// TwinCAT 3 PLC project Untitled1
// ProgramVersion: 3.1.4023.0
// libraries:
//   Tc2_MC2, * (Beckhoff Automation GmbH)
//   Tc2_MC2_Drive, * (Beckhoff Automation GmbH)
//   Tc2_SerialCom, * (Beckhoff Automation GmbH)
//   Tc2_Standard, * (Beckhoff Automation GmbH)
//   Tc2_System, * (Beckhoff Automation GmbH)
//   Tc3_Module, * (Beckhoff Automation GmbH)
// project tree:
//   / ComTask.TcTTO (not stored), PlcTask.TcTTO
//   GVLs/GVLs/ GVL.TcGVL, GVL_IO.TcGVL, GVL_ResearchData.TcGVL, GVL_VAR.TcGVL, ReadMe.TcGVL (not stored)
//   POUs/ FB_Analog.TcPOU, F_ScalAnalogOut.TcPOU, MAIN.TcPOU, P_AP1_Calibrartion.TcPOU, P_ComEL6001.TcPOU (not stored), P_CP1_Enable.TcPOU, P_MI1_OnOff.TcPOU, P_AP1_OnOff.TcPOU, P_Outputs_Manual.TcPOU, P_Set_Research_Data.TcPOU, P_PP1_Ctrl_Manual.TcPOU, P_AP1_Ctrl_Manual.TcPOU, P_Read_Research_Data.TcPOU
//   POUs/POUs/ FB_Drive.TcPOU (not stored), FB_Mixer1_2.TcPOU (not stored)
// real-time tasks:
//   TASK PlcTask: cycle T#10ms, priority 20, ADS port 350
//   TASK ComTask: cycle T#10ms, priority 21, ADS port 351
// motion (NC):
//   TASK NC-Task 1 SAF: cycle T#2ms, priority 4, ADS port 501
//   TASK NC-Task 1 SVB: cycle T#10ms, priority 8, ADS port 511
//   AXIS Mixer 1 (id 2)
//     General: UnitName=°, UnitFlags=#x00000004
//     Dynamic: Acceleration=7443.34, Deceleration=7443.34, Jerk=22330
//     Velo: RefSearch=49.6222741699219, RefSync=49.6222741699219, SlowManual=248.111370849609, FastManual=1488.66822509766, Fast=4962.22741699219, Maximum=4962.23
//     OtherSettings: AllowMotionCmdToSlave=true
//     encoder EncType=8
//       EncPara: ScaleFactorNumerator=45, ScaleFactorDenominator=1048576, Offset=-131121.7408, Inverse=true, MaxCount=#x007fffff, ReferenceSystem=2
//     drive DrvType=9
//       DrvPara: Inverse=true, MaxCount=#xffffffff, DriveControlDWord=#x00030100
//         Analog: VeloReferenz=5458.45015869141, VeloScale=1.02400649589962, ScaleFactorActTorque=0.1
//         TimeComp: TaskDelayCycles=1
//     controller CtrType=1
//       CtrPara: PriorControlFactor=1
//         Observer: BandWidth=20
//   AXIS Mixer 2 (id 3)
//     General: UnitName=°, UnitFlags=#x00000004
//     Dynamic: Acceleration=7443.34112548828, Deceleration=7443.34112548828, Jerk=22330.0233764648
//     Velo: RefSearch=49.6222741699219, RefSync=49.6222741699219, SlowManual=248.111370849609, FastManual=1488.66822509766, Fast=4962.22741699219, Maximum=4962.22741699219
//     OtherSettings: AllowMotionCmdToSlave=true
//     encoder EncType=8
//       EncPara: ScaleFactorNumerator=45, ScaleFactorDenominator=1048576, MaxCount=#x007fffff, ReferenceSystem=2
//     drive DrvType=9
//       DrvPara: MaxCount=#xffffffff, DriveControlDWord=#x00030100
//         Analog: VeloReferenz=5458.45015869141, VeloScale=1.02400649589962, ScaleFactorActTorque=0.1
//         TimeComp: TaskDelayCycles=1
//     controller CtrType=1
//       CtrPara: PriorControlFactor=1
//         Observer: BandWidth=20
// I/O:
//   DEVICE Device 1 (EtherCAT), AmsNetId 172.17.147.1.3.1
//     Term 1 (EK1200) [EK1200-5000 EtherCAT Power supply (2A E-Bus)]
//       Term 2 (EL1008) 30K3 [EL1008 8Ch. Dig. Input 24V, 3ms]
//       Term 3 (EL1008) 30K3.1 [EL1008 8Ch. Dig. Input 24V, 3ms]
//       Term 10 (EL1008) new [EL1008 8Ch. Dig. Input 24V, 3ms]
//       Term 4 (EL2008) 30K4 [EL2008 8Ch. Dig. Output 24V, 0.5A]
//       Term 5 (EL2008) 30K5 [EL2008 8Ch. Dig. Output 24V, 0.5A]
//       Term 12 (EL2008) new [EL2008 8Ch. Dig. Output 24V, 0.5A]
//       Term 13 (EL3022) new [EL3022 2Ch. Ana. Input 4-20mA DIFF]
//       Term 14 (EL3202) new [EL3202 2Ch. Ana. Input PT100 (RTD)]
//       Term 6 (EL3255) 30K5.1 [EL3255 5Ch. potentiometer measurement with sensor supply]
//       Term 7 (EL4134) 30K6 [EL4134 4Ch. Ana. Output -10/+10V, 16bit]
//       Term 8 (EL6001) [EL6001 Interface (RS232)]
//       Term 15 (EL6631) new [EL6631 PROFINET IO Controller]
//       Term 9 (EL9011) [EL9011 End Terminal]
//   DEVICE Device 4 (EtherCAT), AmsNetId 172.17.147.1.5.1
//     Drive 11 (AX5206-0000-0213) [AX5206-0000-0213 EtherCAT Drive (SoE, 2 Ch.)]
// variable links:
//   NC-Task 1 SAF/Axes/Mixer 1 <-> Device 4 (EtherCAT)/Drive 11 (AX5206-0000-0213)
//     Drive/Inputs/In/nDataIn1 <-> AT 1/Following distance
//     Drive/Inputs/In/nDcOutputTime <-> InfoData/DcOutputShift
//     Drive/Inputs/In/nState1 <-> AT 1/Drive status word @bit 8
//     Drive/Inputs/In/nState2 <-> AT 1/Drive status word
//     Drive/Inputs/In/nState4 @bit 1 <-> WcState/InputToggle
//     Drive/Inputs/In/nState4 <-> WcState/WcState
//     Drive/Outputs/Out/nCtrl1 <-> MDT 1/Master control word @bit 8
//     Drive/Outputs/Out/nDataOut1 <-> MDT 1/Position command value
//     Enc/Inputs/In/nDataIn1 <-> AT 1/Position feedback 1 value
//     Enc/Inputs/In/nDcInputTime <-> InfoData/DcInputShift
//     Enc/Inputs/In/nState4 @bit 1 <-> WcState/InputToggle
//     Enc/Inputs/In/nState4 <-> WcState/WcState
//   NC-Task 1 SAF/Axes/Mixer 2 <-> Device 4 (EtherCAT)/Drive 11 (AX5206-0000-0213)
//     Drive/Inputs/In/nDataIn1 <-> AT 2/Following distance
//     Drive/Inputs/In/nDcOutputTime <-> InfoData/DcOutputShift
//     Drive/Inputs/In/nState1 <-> AT 2/Drive status word @bit 8
//     Drive/Inputs/In/nState2 <-> AT 2/Drive status word
//     Drive/Inputs/In/nState4 @bit 1 <-> WcState/InputToggle
//     Drive/Inputs/In/nState4 <-> WcState/WcState
//     Drive/Outputs/Out/nCtrl1 <-> MDT 2/Master control word @bit 8
//     Drive/Outputs/Out/nDataOut1 <-> MDT 2/Position command value
//     Enc/Inputs/In/nDataIn1 <-> AT 2/Position feedback 1 value
//     Enc/Inputs/In/nDcInputTime <-> InfoData/DcInputShift
//     Enc/Inputs/In/nState4 @bit 1 <-> WcState/InputToggle
//     Enc/Inputs/In/nState4 <-> WcState/WcState
//   Untitled1/Untitled1 Instance <-> Device 1 (EtherCAT)/Term 1 (EK1200)/Term 2 (EL1008) 30K3
//     ComTask Inputs/GVL_IO.ib_CC1_Button_Mode_Laptop <-> Channel 8/Input
//     ComTask Inputs/GVL_IO.ib_CP1_Ready <-> Channel 3/Input
//     PlcTask Inputs/GVL_IO.ib_AP1_No_Error <-> Channel 6/Input
//     PlcTask Inputs/GVL_IO.ib_AP1_Ready <-> Channel 5/Input
//     PlcTask Inputs/GVL_IO.ib_CC1_Button_Reset <-> Channel 7/Input
//     PlcTask Inputs/GVL_IO.ib_CC1_Safety_Ready <-> Channel 1/Input
//     PlcTask Inputs/GVL_IO.ib_CP1_Drive_Error <-> Channel 4/Input
//     PlcTask Inputs/GVL_IO.ib_CP1_Safety_Grid_Mounted <-> Channel 2/Input
//   Untitled1/Untitled1 Instance <-> Device 1 (EtherCAT)/Term 1 (EK1200)/Term 3 (EL1008) 30K3.1
//     ComTask Inputs/GVL_IO.ib_PP1_Button_Not_Off <-> Channel 5/Input
//     ComTask Inputs/GVL_IO.ib_PP1_Button_On <-> Channel 4/Input
//     PlcTask Inputs/GVL_IO.ib_AP1_Button_Not_Off <-> Channel 7/Input
//     PlcTask Inputs/GVL_IO.ib_AP1_Button_On <-> Channel 6/Input
//     PlcTask Inputs/GVL_IO.ib_CC1_Button_Mode_Manual <-> Channel 1/Input
//     PlcTask Inputs/GVL_IO.ib_MI1_Button_Not_Off <-> Channel 3/Input
//     PlcTask Inputs/GVL_IO.ib_MI1_Button_On <-> Channel 2/Input
//   Untitled1/Untitled1 Instance <-> Device 1 (EtherCAT)/Term 1 (EK1200)/Term 4 (EL2008) 30K4
//     PlcTask Outputs/GVL_IO.ob_AP1_Pressure_Ok <-> Channel 7/Output
//     PlcTask Outputs/GVL_IO.ob_AP1_Pulse <-> Channel 8/Output
//     PlcTask Outputs/GVL_IO.ob_AP1_Start <-> Channel 6/Output
//     PlcTask Outputs/GVL_IO.ob_CC1_Safety_Reset <-> Channel 1/Output
//     PlcTask Outputs/GVL_IO.ob_CP1_Backward <-> Channel 5/Output
//     PlcTask Outputs/GVL_IO.ob_CP1_Forward <-> Channel 4/Output
//     PlcTask Outputs/GVL_IO.ob_CP1_Start <-> Channel 3/Output
//     PlcTask Outputs/GVL_IO.ob_CP1_Stop <-> Channel 2/Output
//   Untitled1/Untitled1 Instance <-> Device 1 (EtherCAT)/Term 1 (EK1200)/Term 5 (EL2008) 30K5
//     PlcTask Outputs/GVL_IO.ob_AP1_Not_Empty <-> Channel 1/Output
//     PlcTask Outputs/GVL_IO.ob_AP1_Power_On <-> Channel 2/Output
//   Untitled1/Untitled1 Instance <-> Device 1 (EtherCAT)/Term 1 (EK1200)/Term 6 (EL3255) 30K5.1
//     ComTask Inputs/GVL_IO.in_AP1_Poti_Speed <-> AI Standard Channel 3/Value
//     ComTask Inputs/GVL_IO.in_PP1_Poti_Speed <-> AI Standard Channel 2/Value
//     PlcTask Inputs/GVL.nInputSpare1 <-> AI Standard Channel 4/Value
//     PlcTask Inputs/GVL.nInputSpare2 <-> AI Standard Channel 5/Value
//     PlcTask Inputs/GVL_IO.in_MI1_Poti_Speed <-> AI Standard Channel 1/Value
//   Untitled1/Untitled1 Instance <-> Device 1 (EtherCAT)/Term 1 (EK1200)/Term 7 (EL4134) 30K6
//     PlcTask Outputs/GVL_IO.on_AP1_Speed <-> AO Output Channel 2/Analog output
//     PlcTask Outputs/GVL_IO.on_CP1_Speed <-> AO Output Channel 1/Analog output
//   Untitled1/Untitled1 Instance <-> Device 1 (EtherCAT)/Term 1 (EK1200)/Term 8 (EL6001)
//     ComTask Inputs/GVL.stIn_EL6001/D <-> COM Inputs/Data In 0
//     ComTask Inputs/GVL.stIn_EL6001/D @bit {8..168 step 8} <-> COM Inputs/Data In {1..21}  (21 links)
//     ComTask Inputs/GVL.stIn_EL6001/Status <-> COM Inputs/Status
//     ComTask Outputs/GVL.stOut_EL6001/Ctrl <-> COM Outputs/Ctrl
//     ComTask Outputs/GVL.stOut_EL6001/D <-> COM Outputs/Data Out 0
//     ComTask Outputs/GVL.stOut_EL6001/D @bit {8..168 step 8} <-> COM Outputs/Data Out {1..21}  (21 links)
//   Untitled1/Untitled1 Instance <-> Device 4 (EtherCAT)/Drive 11 (AX5206-0000-0213)
//     PlcTask Inputs/GVL.in_MID1_ActAbsCurrent <-> AT 1/Actual absolute current
//     PlcTask Inputs/GVL.in_MID2_ActAbsCurrent <-> AT 2/Actual absolute current
//     PlcTask Inputs/GVL.in_MID1_ActMotorTemperature <-> AT 1/Motor temperature
//     PlcTask Inputs/GVL.in_MID2_ActMotorTemperature <-> AT 2/Motor temperature
//   Untitled1/Untitled1 Instance <-> NC-Task 1 SAF/Axes/Mixer 1
//     PlcTask Inputs/GVL.Axis_Mixer1.NcToPlc <-> Outputs/ToPlc
//     PlcTask Outputs/GVL.Axis_Mixer1.PlcToNc <-> Inputs/FromPlc
//   Untitled1/Untitled1 Instance <-> NC-Task 1 SAF/Axes/Mixer 2
//     PlcTask Inputs/GVL.Axis_Mixer2.NcToPlc <-> Outputs/ToPlc
//     PlcTask Outputs/GVL.Axis_Mixer2.PlcToNc <-> Inputs/FromPlc

CONFIGURATION Untitled1
    RESOURCE PLC ON TwinCAT3
        TASK PlcTask(INTERVAL := T#10ms, PRIORITY := 20);
        PROGRAM MAIN WITH PlcTask : MAIN;
    END_RESOURCE
END_CONFIGURATION

// ---- GVLs/GVLs/GVL.TcGVL
{attribute 'qualified_only'}
VAR_GLOBAL
	
	
	//
	// Data Communication RS-232
	TxBufferEL								: ComBuffer;
	RxBufferEL								: ComBuffer;
	
			
	//
	// Data Communication Axis Mixers

	//
	// Mixer drive A // 16.09.2021 PF
	Axis_Mixer1 							: AXIS_REF;
	f_MID1_ActCurrent: REAL;
	f_MID1_ActTorque: REAL;
	in_MID1_ActAbsCurrent AT %I*: INT;
	in_MID1_ActMotorTemperature AT %I* :INT; // 220817 weiting added
	
	//
	// Mixer drive B // 16.09.2021 PF
	Axis_Mixer2 							: AXIS_REF;
	f_MID2_ActCurrent: REAL;
	f_MID2_ActTorque: REAL;
	in_MID2_ActAbsCurrent AT %I*: INT;
	in_MID2_ActMotorTemperature AT %I* :INT; // 220817 weiting added
	
	//
	// Control Input Speed
	fControlMixerPumpSpeed					: REAL; 
	fControlPeristalticPumpSpeed			: REAL; 
	fControlDosingPumpSpeed					: REAL; 
	fInputSpare1							: REAL; 
	fInputSpare2							: REAL; 
	
	//
	// Output Speed
	fConcretePumpSpeed						: REAL;
	fDosingPumpSpeed						: REAL;
	fOutputSpare1							: REAL;
	fOutputSpare2							: REAL;
	
	
	//
	//Hardware Input
	bSafetyIO						AT %I*	: BOOL;
	// bConcretePumpSafetyGridMounted	AT %I*	: BOOL;
	// bConcretePumpReady				AT %I*	: BOOL;
	// bConcretePumpFcError				AT %I*	: BOOL;
	bDosingPumpReady				AT %I*	: BOOL;
	bDosingPumpNoError				AT %I*	: BOOL;
	bControlResetSafety				AT %I*	: BOOL;
	bControlLaptop					AT %I*	: BOOL;
	bControlManual					AT %I*	: BOOL;	
	nControlMixerPumpOn				AT %I*	: BOOL; 
	nControlMixerPumpOff			AT %I*	: BOOL; 
	nControlConcretPumpOn			AT %I*	: BOOL; 
	nControlConcretPumpOff			AT %I*	: BOOL; 
	nControlDosingPumpOn			AT %I*	: BOOL; 
	nControlDosingPumpOff			AT %I*	: BOOL; 
	bInputSpare1					AT %I*	: BOOL;
		
	nControlMixerPumpSpeed			AT %I*	: INT; 
	// nControlPeristalticPumpSpeed	AT %I*	: INT; 
	nControlDosingPumpSpeed			AT %I*	: INT; 
	nInputSpare1					AT %I*	: INT; 
	nInputSpare2					AT %I*	: INT; 

	
	//
	//Hardware Output
	bResetSafety					AT %Q*	: BOOL;
	// bConcretePumpOn					AT %Q*	: BOOL;
	// bConcretePumpOff					AT %Q*	: BOOL;
	// bConcretePumpForwardOn			AT %Q*	: BOOL;
	// bConcretePumpBackwardOn			AT %Q*	: BOOL;
	bDosingPumpDosingHighLow		AT %Q*	: BOOL;
	bDosingPumpNoFastStop			AT %Q*	: BOOL;
	bDosingPumpDosingAmount			AT %Q*	: BOOL;
	bOutputSpare1					AT %Q*	: BOOL;
	bOutputSpare2					AT %Q*	: BOOL;
	bOutputSpare3					AT %Q*	: BOOL;
	bOutputSpare4					AT %Q*	: BOOL;
	bOutputSpare5					AT %Q*	: BOOL;
	bOutputSpare6					AT %Q*	: BOOL;
	bOutputSpare7					AT %Q*	: BOOL;
	bOutputSpare8					AT %Q*	: BOOL;
	
	// nConcretePumpSpeed				AT %Q*	: INT;
	nDosingPumpSpeed				AT %Q*	: INT;
	nOutputSpare1					AT %Q*	: INT;
	nOutputSpare2					AT %Q*	: INT;
	
	
	//
	//Hardware RS-232
	stIn_EL6001 					AT %I*	: EL6inData22B;	
	stOut_EL6001 					AT %Q*	: EL6outData22B;
	
END_VAR

// ---- GVLs/GVLs/GVL_IO.TcGVL
{attribute 'qualified_only'}
VAR_GLOBAL
//***********************************************************************************
//
// ETH Zürich / Robotic Fabrication Lab
// HIB C 13 / Stefano-Franscini-Platz 1
// CH-8093 Zürich
// 
// ***********************************************************************************
// 
// PROJECT     :  A061 Inline Mixer
// 
// FUNCTION    :  Global Varable In and Outputs
// 
// AUTHOR      :  Fabio Scotto / Philippe Fleischmann
// 
// EMAIL       :  scotto@arch.ethz.ch / fleischmann@arch.ehtz.ch
// 
// Copyright   :  ETH Zürich (CH) 2020
//
// ***********************************************************************************

//
// Inputs

//
// Concrete Controller 1
ib_CC1_Safety_Ready AT %I*: BOOL;
ib_CC1_Button_Mode_Manual AT %I*: BOOL;
ib_CC1_Button_Mode_Laptop AT %I*: BOOL;
ib_CC1_Button_Reset AT %I*: BOOL;
//
// Concrete Pump 1
ib_CP1_Drive_Error AT %I*: BOOL;
ib_CP1_Ready AT %I*: BOOL;
ib_CP1_Safety_Grid_Mounted AT %I*: BOOL;
in_CP1_Tube_Pressure_Sensor AT %I*: INT;
in_CP1_Tube_Temperature_Sensor AT %I*: INT;

//
// Peristaltic Pump 1
ib_PP1_Button_On AT %I*: BOOL;
ib_PP1_Button_Not_Off AT %I*: BOOL;
in_PP1_Poti_Speed AT %I*	: INT; 

//
// Accelerator Pump 1
ib_AP1_Button_On AT %I*: BOOL;
ib_AP1_Button_Not_Off AT %I*: BOOL;
ib_AP1_Ready AT %I*: BOOL;
ib_AP1_No_Error AT %I*: BOOL;
in_AP1_Poti_Speed AT %I*	: INT; 

//
// Mixer 1
ib_MI1_Button_On AT %I*: BOOL;
ib_MI1_Button_Not_Off AT %I*: BOOL;
in_MI1_Poti_Speed AT %I*	: INT; 

//
// Outputs

//
// Concrete Controller 1
ob_CC1_Safety_Reset AT %Q*: BOOL;

//
// Concrete Pump 1
ob_CP1_Start AT %Q*: BOOL;
ob_CP1_Stop AT %Q*: BOOL;
ob_CP1_Forward AT %Q*: BOOL;
ob_CP1_Backward AT %Q*: BOOL;

on_CP1_Speed AT %Q*: INT;

//
// Accelerator Pump 1
ob_AP1_Power_On AT %Q*: BOOL;
ob_AP1_Start AT %Q*: BOOL;
ob_AP1_Pressure_Ok AT %Q*: BOOL;
ob_AP1_Not_Empty AT %Q*: BOOL;
ob_AP1_Pulse AT %Q*: BOOL;

on_AP1_Speed AT %Q*: INT;


END_VAR

// ---- GVLs/GVLs/GVL_ResearchData.TcGVL
{attribute 'qualified_only'}
VAR_GLOBAL
//***********************************************************************************
//
// ETH Zürich / Robotic Fabrication Lab
// HIB C 13 / Stefano-Franscini-Platz 1
// CH-8093 Zürich
// 
// ***********************************************************************************
// 
// PROJECT     :  A061 Inline Mixer
// 
// FUNCTION    :  Global Varable to collect all research data
// 
// AUTHOR      :  Seyma Gürel / Philippe Fleischmann
// 
// EMAIL       :  scotto@arch.ethz.ch / fleischmann@arch.ehtz.ch
// 
// Copyright   :  ETH Zürich (CH) 2021
//
// ***********************************************************************************


// ***********************************************************************************
// Process inputs
// ***********************************************************************************

//
// Maximal speed for mixer [°/s]  
f_RED_Control_Speed : LREAL;					// [°/s]

//
// Accelerator Pump
b_RED_Acceleration_Pump_Calibration_On: BOOL;
n_RED_Acceleration_Pump_Calibration_Speed: INT;
n_RED_Acceleration_Pump_Calibration_Time: TIME;
f_RED_Acceleration_Pump_Mass: REAL;             // [g/min]
f_RED_Acceleration_Pump_Density: REAL;          // [g/ml]
n_RED_Acceleration_Pump_Flowrate: REAL;         // [ml/min]

//
// Concrete Pump
b_RED_Concrete_Pump_Forward_On: BOOL;
b_RED_Concrete_Pump_Backward_On: BOOL;
n_RED_Concrete_Pump_Speed: INT;					// [ 0..75rpm ]
		

// ***********************************************************************************
// Process outpus
// ***********************************************************************************

//
// Status mixer
b_RED_Status_On : BOOL;
f_RED_Status_Speed_Overide : LREAL;
f_RED_Status_Speed_Motor_1 : LREAL;
f_RED_Status_Speed_Motor_2 : LREAL;
f_RED_Status_Torque_Motor_1 : REAL;				// [Nm]
f_RED_Status_Torque_Motor_2 : REAL;				// [Nm]

// Weiting added 220817 
f_RED_Status_Temperature_Motor_1 : REAL; // [°C] 
f_RED_Status_Temperature_Motor_2 : REAL; // [°C] 

//
// Accelerator Pump
n_RED_Status_Acceleration_Pump_Flowrate: INT;          // [ml/min]
f_RED_Status_Acceleration_Pump_Max_Flowrate_ml_per_min: REAL;           // [ml/min]

END_VAR

// ---- GVLs/GVLs/GVL_VAR.TcGVL
{attribute 'qualified_only'}
VAR_GLOBAL
//***********************************************************************************
//
// ETH Zürich / Robotic Fabrication Lab
// HIB C 13 / Stefano-Franscini-Platz 1
// CH-8093 Zürich
// 
// ***********************************************************************************
// 
// PROJECT     :  A061 Inline Mixer
// 
// FUNCTION    :  Global Varable In and Outputs
// 
// AUTHOR      :  Fabio Scotto / Philippe Fleischmann
// 
// EMAIL       :  scotto@arch.ethz.ch / fleischmann@arch.ehtz.ch
// 
// Copyright   :  ETH Zürich (CH) 2020
//
// ***********************************************************************************

//
// Concrete Controller 1

//
// Concrete Pump 1

//
// Peristaltic Pump 1

//
// Accelerator Pump 1
b_AP1_Run : BOOL;
f_AP1_Override : LREAL; 

//
// Mixer 1
b_MI1_ReadToDrive : BOOL;
b_MI1_Run : BOOL;
f_MI1_Override : LREAL; 
f_MI1_MaxSpeed : LREAL;
f_MI1_ActSpeedM1 : LREAL;
f_MI1_ActSpeedM2 : LREAL;

END_VAR

// ---- POUs/MAIN.TcPOU
PROGRAM MAIN
VAR	

	fb_MC_SetPosition		:FB_SoEAX5000SetPositionOffset;
	pos:real;
	Mixer1_2		: FB_Mixer1_2;
	Analog			: FB_Analog;

	SafetyReset 	: bool;
	b_Enable		: BOOL;
	b_Reset			: BOOL;


	
	Test : MC_ReadStatus;
END_VAR

//***********************************************************************************
//
// ETH Zürich / Robotic Fabrication Lab
// HIB C 13 / Stefano-Franscini-Platz 1
// CH-8093 Zürich
// 
// ***********************************************************************************
// 
// PROJECT     :  A061 Inline Mixer
// 
// FUNCTION    :  MAIN Programm
// 
// AUTHOR      :  Mathias Suter
// 
// EMAIL       :  mathias.suter@solinaut.ch
// 
// Copyright   :  ETH Zürich (CH) 2021
//
// ***********************************************************************************


//
// Mode selector 
//P_ModeSelector();

//
// Set research data 
P_Set_Research_Data();

//
// Acceleration Pump 1 On/off 
P_AP1_Calibrartion();

//
// Check for Acceleration Pump 1 state
IF GVL_ResearchData.b_RED_Acceleration_Pump_Calibration_On=FALSE THEN
	//
	// Acceleration Pump 1 On/off 
	P_AP1_OnOff();
END_IF

//
// Temporary scaling of the poti for the mixer override  
GVL_VAR.f_MI1_Override:=100.0 / 32767 * GVL_IO.in_MI1_Poti_Speed;

//
// Peristaltic Pump 1 manual control 
//P_PP1_Ctrl_Manual();

//
// Mixer On/Off 
P_MI1_OnOff();

//
// Temporary scaling of the poti for the mixer override  
GVL_VAR.f_MI1_Override:=100.0 / 32767 * GVL_IO.in_MI1_Poti_Speed;

//
// Mixer 1 + 2
Mixer1_2(
	Mixer1			:= GVL.Axis_Mixer1,
 	Mixer2			:= GVL.Axis_Mixer2,
	f_Velocity		:= GVL_VAR.f_MI1_MaxSpeed,
	b_JogForward	:= FALSE,
	b_JogBackwards	:= GVL_VAR.b_MI1_Run,
 	b_Enable		:= GVL_IO.ib_CC1_Button_Mode_Manual AND GVL_IO.ib_CC1_Safety_Ready,	
 	b_Reset			:= GVL_IO.ib_CC1_Button_Reset,
	f_Override		:= GVL_VAR.f_MI1_Override);	
	(*
	fb_MC_SetPosition(
	Axis			:= GVL.Axis_Mixer2,
	memory			:= 1,
	Feedback		:= 0);*)
	
pos:=GVL.Axis_Mixer2.NcToPlc.ModuloActPos;


//
GVL.f_MID1_ActCurrent:=GVL.in_MID1_ActAbsCurrent * 5.9 / 1000;
GVL.f_MID1_ActTorque:=GVL.f_MID1_ActCurrent * 1.4 * 8; // Torque constante / Gear transaltion

GVL.f_MID2_ActCurrent:=gvl.in_MID2_ActAbsCurrent * 5.9 / 1000;
GVL.f_MID2_ActTorque:=GVL.f_MID2_ActCurrent * 1.4 * 8; // Torque constante / Gear transaltion

//
// Write global variable for mixer ready to drive
GVL_VAR.b_MI1_ReadToDrive:=Mixer1_2.b_ReadyToDrive;
	
// 
// Reset 
GVL_IO.ob_CC1_Safety_Reset:=GVL_IO.ib_CC1_Button_Reset;
 	
// GVL.bResetSafety	:= safetyReset;


//
// Concrete pump
P_CP1_Enable();
	
// Analog();

//
// Outputs
P_Outputs_Manual();

//
// Read researchs data 
P_Read_Research_Data();

END_PROGRAM

// ---- POUs/FB_Analog.TcPOU
FUNCTION_BLOCK FB_Analog
VAR_INPUT
END_VAR
VAR_OUTPUT
END_VAR
VAR
END_VAR

//***********************************************************************************
//
// ETH Zürich / Robotic Fabrication Lab
// HIB C 13 / Stefano-Franscini-Platz 1
// CH-8093 Zürich
// 
// ***********************************************************************************
// 
// PROJECT     :  ?? 
// 
// FUNCTION    :  Analog Calculation
// 
// AUTHOR      :  Mathias Suter
// 
// EMAIL       :  mathias.suter@solinaut.ch
// 
// Copyright   :  ETH Zürich (CH) 2021
//
// ***********************************************************************************


//
// Analog Inputs - Scale 0-100%
GVL.fControlMixerPumpSpeed := INT_TO_REAL(GVL.nControlMixerPumpSpeed) / 32767 * 100;			
//GVL.fControlPeristalticPumpSpeed := INT_TO_REAL(GVL.nControlPeristalticPumpSpeed) / 32767 * 100;			
GVL.fControlDosingPumpSpeed := INT_TO_REAL(GVL.nControlDosingPumpSpeed) / 32767 * 100;				
GVL.fInputSpare1 := INT_TO_REAL(GVL.nInputSpare1) / 32767 * 100;						
GVL.fInputSpare2 := INT_TO_REAL(GVL.nInputSpare2) / 32767 * 100;						
	

//
// Analog Outputs - Scale 0-100%
// GVL.nConcretePumpSpeed := REAL_TO_INT(GVL.fConcretePumpSpeed / 100 * 32767);				
GVL.nDosingPumpSpeed := REAL_TO_INT(GVL.fDosingPumpSpeed / 100 * 32767);					
GVL.nOutputSpare1 := REAL_TO_INT(GVL.fOutputSpare1 / 100 * 32767);						
GVL.nOutputSpare2 := REAL_TO_INT(GVL.fOutputSpare2 / 100 * 32767);

END_FUNCTION_BLOCK

// ---- POUs/P_Set_Research_Data.TcPOU
PROGRAM P_Set_Research_Data
VAR


END_VAR

//***********************************************************************************
//
// ETH Zürich / Robotic Fabrication Lab
// HIB C 13 / Stefano-Franscini-Platz 1
// CH-8093 Zürich
// 
// ***********************************************************************************
// 
// PROJECT     :  A061 Inline Mixer
// 
// FUNCTION    :  Set all research data for the process
// 
// AUTHOR      :  Seyma Gürel / Philippe Fleischmann
// 
// EMAIL       :  scotto@arch.ethz.ch / fleischmann@arch.ehtz.ch
// 
// Copyright   :  ETH Zürich (CH) 2021
//
// ***********************************************************************************


//
// Updating Mixer 1 max speed [°/s]
GVL_ResearchData.f_RED_Control_Speed:=720;
GVL_VAR.f_MI1_MaxSpeed:=GVL_ResearchData.f_RED_Control_Speed;

//
// Updating Acceleration Pump calibration values 
GVL_ResearchData.n_RED_Acceleration_Pump_Calibration_Speed:=32767;     // [raw date]
GVL_ResearchData.n_RED_Acceleration_Pump_Calibration_Time:=T#60000MS;   // [ms]
//GVL_ResearchData.f_RED_Acceleration_Pump_Mass:=342.0;                    // [g/min]
GVL_ResearchData.f_RED_Acceleration_Pump_Density:=2.047;               // [g/ml]

END_PROGRAM

// ---- POUs/P_AP1_Calibrartion.TcPOU
PROGRAM P_AP1_Calibrartion
VAR_INPUT
	//
	// INT 
	n_Step: INT := 0;	
END_VAR
VAR
	//
	// BOOL 
	b_Condition: BOOL;

	//
	// Timer
	t_AP1_Calibration_Time: TON; 
	
END_VAR

//***********************************************************************************
//
// ETH Zürich / Robotic Fabrication Lab
// HIB C 13 / Stefano-Franscini-Platz 1
// CH-8093 Zürich
// 
// ***********************************************************************************
// 
// PROJECT     :  A061 Inline Mixer
// 
// FUNCTION    :  Step chain for accelerator pump calibration
// 
// AUTHOR      :  Seyma Gürel / Philippe Fleischmann
// 
// EMAIL       :  sguerel@ethz.ch / fleischmann@arch.ehtz.ch
// 
// Copyright   :  ETH Zürich (CH) 2021
//
// ***********************************************************************************

//
// Initalization
IF n_Step=0 THEN
	//
	// Check condition 
	b_Condition:=TRUE;
	//
	// Do step
	IF b_Condition THEN
		b_Condition:=FALSE;
		n_Step:=10;
	END_IF
END_IF

//
// Wait for activating calibration
IF n_Step=10 THEN
	//
	// Check condition 
	b_Condition:= GVL_ResearchData.b_RED_Acceleration_Pump_Calibration_On;
	//
	// Do step
	IF b_Condition THEN
		b_Condition:=FALSE;
		n_Step:=20;
	END_IF
END_IF

//
// Wait for start 
IF n_Step=20 THEN
	//
	// Check condition 
	b_Condition:=GVL_IO.ib_AP1_Button_On;
	//
	// Do step
	IF b_Condition THEN
		b_Condition:=FALSE;
		n_Step:=30;
	END_IF
END_IF

//
// Run calibration until time is over 
IF n_Step=30 THEN
	//
	// Check condition 
	b_Condition:=t_AP1_Calibration_Time.Q; 
	//
	// Do step
	IF b_Condition THEN
		b_Condition:=FALSE;
		n_Step:=40;
	END_IF
END_IF

//
// Return to step 10 
IF n_Step=40 THEN
	//
	// Check condition 
	b_Condition:=TRUE;
	//
	// Do step
	IF b_Condition THEN
		b_Condition:=FALSE;
		//
		// Reset calibrarion on
		GVL_ResearchData.b_RED_Acceleration_Pump_Calibration_On:=FALSE;
		n_Step:=10;
	END_IF
END_IF

// ****************************************
// Timer
// ****************************************
t_AP1_Calibration_Time(
	IN:=n_Step=30,
	PT:=GVL_ResearchData.n_RED_Acceleration_Pump_Calibration_Time);

// ****************************************
// Reset
// ****************************************

IF GVL_ResearchData.b_RED_Acceleration_Pump_Calibration_On=FALSE THEN
  //
  // Rest step chain
  n_Step:=0;
END_IF

END_PROGRAM

// ---- POUs/P_AP1_OnOff.TcPOU
PROGRAM P_AP1_OnOff
VAR_INPUT
	//
	// INT 
	n_Step: INT := 0;	
END_VAR
VAR
	//
	// BOOL 
	b_Condition: BOOL;
	b_No_Emergency_Stop:BOOL :=TRUE;
	
END_VAR

//***********************************************************************************
//
// ETH Zürich / Robotic Fabrication Lab
// HIB C 13 / Stefano-Franscini-Platz 1
// CH-8093 Zürich
// 
// ***********************************************************************************
// 
// PROJECT     :  A061 Inline Mixer
// 
// FUNCTION    :  Step chain for accelerator pump on or off 
// 
// AUTHOR      :  Fabio Scotto / Philippe Fleischmann
// 
// EMAIL       :  scotto@arch.ethz.ch / fleischmann@arch.ehtz.ch
// 
// Copyright   :  ETH Zürich (CH) 2020
//
// ***********************************************************************************

//
// Ignore emergency stop
b_No_Emergency_Stop:=TRUE;

//
// Initalization
IF n_Step=0 THEN
	//
	// Check condition 
	b_Condition:=TRUE;
	//
	// Do step
	IF b_Condition THEN
		b_Condition:=FALSE;
		n_Step:=10;
	END_IF
END_IF

//
// Wait for start mixer
IF n_Step=10 THEN
	//
	// Check condition 
	b_Condition:= GVL_IO.ib_AP1_Ready AND GVL_IO.ib_AP1_Button_On;
	//
	// Do step
	IF b_Condition AND b_No_Emergency_Stop THEN
		b_Condition:=FALSE;
		n_Step:=20;
	END_IF
END_IF

//
// Reserve
IF n_Step=20 THEN
	//
	// Check condition 
	b_Condition:=TRUE;
	//
	// Do step
	IF b_Condition AND b_No_Emergency_Stop THEN
		b_Condition:=FALSE;
		n_Step:=30;
	END_IF
END_IF

//
// Run for mixer 
IF n_Step=30 THEN
	//
	// Check condition 
	b_Condition:= NOT GVL_IO.ib_AP1_Button_Not_Off OR NOT GVL_IO.ib_AP1_No_Error ;
	//
	// Do step
	IF b_Condition THEN
		b_Condition:=FALSE;
		n_Step:=40;
	END_IF
END_IF

//
// Reserve
IF n_Step=40 THEN
	//
	// Check condition 
	b_Condition:=TRUE;
	//
	// Do step
	IF b_Condition AND b_No_Emergency_Stop THEN
		b_Condition:=FALSE;
		n_Step:=50;
	END_IF
END_IF

//
// Return to step 10 
IF n_Step=50 THEN
	//
	// Check condition 
	b_Condition:=TRUE;
	//
	// Do step
	IF b_Condition THEN
		b_Condition:=FALSE;
		n_Step:=10;
	END_IF
END_IF

// ****************************************
// Write global variabls
// ****************************************

//
// Mixer run
GVL_VAR.b_AP1_Run:=n_Step=30;


// ****************************************
// Timer
// ****************************************

END_PROGRAM

// ---- POUs/P_MI1_OnOff.TcPOU
PROGRAM P_MI1_OnOff
VAR_INPUT
	//
	// INT 
	n_Step: INT := 0;	
END_VAR
VAR
	//
	// BOOL 
	b_Condition: BOOL;
	b_No_Emergency_Stop:BOOL :=TRUE;
	
END_VAR

//***********************************************************************************
//
// ETH Zürich / Robotic Fabrication Lab
// HIB C 13 / Stefano-Franscini-Platz 1
// CH-8093 Zürich
// 
// ***********************************************************************************
// 
// PROJECT     :  A061 Inline Mixer
// 
// FUNCTION    :  Step chain for mixer on or off 
// 
// AUTHOR      :  Fabio Scotto / Philippe Fleischmann
// 
// EMAIL       :  scotto@arch.ethz.ch / fleischmann@arch.ehtz.ch
// 
// Copyright   :  ETH Zürich (CH) 2020
//
// ***********************************************************************************

// Ignore emergency stop
b_No_Emergency_Stop:=TRUE;

//
// Initalization
IF n_Step=0 THEN
	//
	// Check condition 
	b_Condition:=TRUE;
	//
	// Do step
	IF b_Condition THEN
		b_Condition:=FALSE;
		n_Step:=10;
	END_IF
END_IF

//
// Wait for start mixer
IF n_Step=10 THEN
	//
	// Check condition 
	b_Condition:= GVL_VAR.b_MI1_ReadToDrive AND GVL_IO.ib_MI1_Button_On;
	//
	// Do step
	IF b_Condition AND b_No_Emergency_Stop THEN
		b_Condition:=FALSE;
		n_Step:=20;
	END_IF
END_IF

//
// Reserve
IF n_Step=20 THEN
	//
	// Check condition 
	b_Condition:=TRUE;
	//
	// Do step
	IF b_Condition AND b_No_Emergency_Stop THEN
		b_Condition:=FALSE;
		n_Step:=30;
	END_IF
END_IF

//
// Run for mixer 
IF n_Step=30 THEN
	//
	// Check condition 
	b_Condition:= NOT GVL_IO.ib_MI1_Button_Not_Off OR NOT GVL_VAR.b_MI1_ReadToDrive;
	//
	// Do step
	IF b_Condition THEN
		b_Condition:=FALSE;
		n_Step:=40;
	END_IF
END_IF

//
// Reserve
IF n_Step=40 THEN
	//
	// Check condition 
	b_Condition:=TRUE;
	//
	// Do step
	IF b_Condition AND b_No_Emergency_Stop THEN
		b_Condition:=FALSE;
		n_Step:=50;
	END_IF
END_IF

//
// Return to step 10 
IF n_Step=50 THEN
	//
	// Check condition 
	b_Condition:=TRUE;
	//
	// Do step
	IF b_Condition THEN
		b_Condition:=FALSE;
		n_Step:=10;
	END_IF
END_IF

// ****************************************
// Write global variabls
// ****************************************

//
// Mixer run
GVL_VAR.b_MI1_Run:=n_Step=30;


// ****************************************
// Timer
// ****************************************

END_PROGRAM

// ---- POUs/P_CP1_Enable.TcPOU
PROGRAM P_CP1_Enable
VAR_INPUT
	//
	// INT 
	n_Step: INT := 0;	
END_VAR
VAR
	//
	// BOOL 
	b_Condition: BOOL;
	b_No_Emergency_Stop:BOOL :=TRUE;

	//
	// Timer 
	t_CP1_Puls_Enable: TON;	
	t_CP1_Puls_Disable: TON;	
	
END_VAR

//***********************************************************************************
//
// ETH Zürich / Robotic Fabrication Lab
// HIB C 13 / Stefano-Franscini-Platz 1
// CH-8093 Zürich
// 
// ***********************************************************************************
// 
// PROJECT     :  A059 Aero Crete 
// 
// FUNCTION    :  Step chain for concrete pump enable 
// 
// AUTHOR      :  Nicolas Feihl / Philippe Fleischmann
// 
// EMAIL       :  feihl@arch.ethz.ch / fleischmann@arch.ehtz.ch
// 
// Copyright   :  ETH Zürich (CH) 2020
//
// ***********************************************************************************

// Ignore emergency stop
b_No_Emergency_Stop:=TRUE;

//
// Initalization
IF n_Step=0 THEN
	//
	// Check condition 
	b_Condition:=TRUE;
	//
	// Do step
	IF b_Condition THEN
		b_Condition:=FALSE;
		n_Step:=10;
	END_IF
END_IF

//
// Check grid mounted and no errors 
IF n_Step=10 THEN
	//
	// Check condition 
	b_Condition:= GVL_IO.ib_CP1_Safety_Grid_Mounted AND NOT GVL_IO.ib_CP1_Drive_Error;
	//
	// Do step
	IF b_Condition AND b_No_Emergency_Stop THEN
		b_Condition:=FALSE;
		n_Step:=20;
	END_IF
END_IF

//
// Send enable to pump
IF n_Step=20 THEN
	//
	// Check condition 
	b_Condition:=t_CP1_Puls_Enable.Q;
	//
	// Do step
	IF b_Condition AND b_No_Emergency_Stop THEN
		b_Condition:=FALSE;
		n_Step:=30;
	END_IF
END_IF

//
// Pump enabled checking for errors or grid removed
IF n_Step=30 THEN
	//
	// Check condition 
	b_Condition:= NOT GVL_IO.ib_CP1_Safety_Grid_Mounted OR GVL_IO.ib_CP1_Drive_Error;
	//
	// Do step
	IF b_Condition THEN
		b_Condition:=FALSE;
		n_Step:=40;
	END_IF
END_IF

//
// Send disable to pump
IF n_Step=40 THEN
	//
	// Check condition 
	b_Condition:=t_CP1_Puls_Disable.Q;
	//
	// Do step
	IF b_Condition AND b_No_Emergency_Stop THEN
		b_Condition:=FALSE;
		n_Step:=50;
	END_IF
END_IF

//
// Return to step 10 
IF n_Step=50 THEN
	//
	// Check condition 
	b_Condition:=TRUE;
	//
	// Do step
	IF b_Condition THEN
		b_Condition:=FALSE;
		n_Step:=10;
	END_IF
END_IF

// ****************************************
// Timer
// ****************************************
t_CP1_Puls_Enable(
	IN:=n_Step=20,
	PT:=T#200MS);

t_CP1_Puls_Disable(
	IN:=n_Step=40,
	PT:=T#200MS);

END_PROGRAM

// ---- POUs/P_Outputs_Manual.TcPOU
PROGRAM P_Outputs_Manual
VAR


END_VAR

//***********************************************************************************
//
// ETH Zürich / Robotic Fabrication Lab
// HIB C 13 / Stefano-Franscini-Platz 1
// CH-8093 Zürich
// 
// ***********************************************************************************
// 
// PROJECT     :  A061 Inline Mixer
// 
// FUNCTION    :  Outputs Manual Mode
// 
// AUTHOR      :  Fabio Scotto / Philippe Fleischmann
// 
// EMAIL       :  scotto@arch.ethz.ch / fleischmann@arch.ehtz.ch
// 
// Copyright   :  ETH Zürich (CH) 2020
//
// ***********************************************************************************


//
// Accelerator pump 1

//
// Power on
GVL_IO.ob_AP1_Power_On:=GVL_IO.ib_CC1_Button_Mode_Manual;

//
// Pressure okey always set to true
GVL_IO.ob_AP1_Pressure_Ok:=TRUE;

//
// Bucket not empty always set to true
GVL_IO.ob_AP1_Not_Empty:=TRUE;

//
// Pulse a preset amount not in use
GVL_IO.ob_AP1_Pulse:=FALSE;

//
// Start pump
IF 	   P_AP1_OnOff.n_Step=30 
	OR P_AP1_Calibrartion.n_Step=30
THEN
	//
	// Pump on
	GVL_IO.ob_AP1_Start:=TRUE;
ELSE
	//
	// Pump off
	GVL_IO.ob_AP1_Start:=FALSE;
END_IF

//
// Speed for pump
IF 	   P_AP1_Calibrartion.n_Step=20 
	OR P_AP1_Calibrartion.n_Step=30 
THEN
	//
	// Calibration Speed for pump
	GVL_IO.on_AP1_Speed:=GVL_ResearchData.n_RED_Acceleration_Pump_Calibration_Speed;
ELSE
	//
	// Process speed for pump
	GVL_IO.on_AP1_Speed:=F_ScalAnalogOut(
		n_Input:= REAL_TO_INT(GVL_ResearchData.n_RED_Acceleration_Pump_Flowrate),
		n_InMin:= 0, 
		n_InMax:= REAL_TO_INT(GVL_ResearchData.f_RED_Status_Acceleration_Pump_Max_Flowrate_ml_per_min), 
		n_OutMin:= 0, 
		n_OutMax:= 32767);
END_IF

// ***********************************************************************************
// Concrete Pump 1 
// ***********************************************************************************

//
// Start
IF  P_CP1_Enable.n_Step=20 THEN
	GVL_IO.ob_CP1_Start:=TRUE;
ELSE
	GVL_IO.ob_CP1_Start:=FALSE;
END_IF

//
// Stop
IF  P_CP1_Enable.n_Step=40 THEN
	GVL_IO.ob_CP1_Stop:=TRUE;
ELSE
	GVL_IO.ob_CP1_Stop:=FALSE;
END_IF

//
// Forward
GVL_IO.ob_CP1_Forward:=GVL_ResearchData.b_RED_Concrete_Pump_Forward_On;

//
// Backward
GVL_IO.ob_CP1_Backward:=GVL_ResearchData.b_RED_Concrete_Pump_Backward_On;

//
// Concrete pump speed  0 (0V) to 75 rpm (10V)
GVL_IO.on_CP1_Speed:=F_ScalAnalogOut(
	n_Input:=GVL_ResearchData.n_RED_Concrete_Pump_Speed, 
	n_InMin:=0, 
	n_InMax:=75, 
	n_OutMin:=0, 
	n_OutMax:=32767);

END_PROGRAM

// ---- POUs/F_ScalAnalogOut.TcPOU
FUNCTION F_ScalAnalogOut : INT
VAR_INPUT
	n_Input:INT;
	n_InMin:INT;
	n_InMax:INT;
	n_OutMin:INT;
	n_OutMax:INT;

END_VAR
VAR
	f_Input:REAL;
	f_InMin:REAL;
	f_InMax:REAL;
	f_OutMin:REAL;
	f_OutMax:REAL;
	f_DeltaIn:REAL;
	f_DeltaOut:REAL;
END_VAR

//
// Convert integer to real 
f_Input:=INT_TO_REAL(n_Input);
f_InMin:=INT_TO_REAL(n_InMin);
f_InMax:=INT_TO_REAL(n_InMax);
f_OutMin:=INT_TO_REAL(n_OutMin);
f_OutMax:=INT_TO_REAL(n_OutMax);
//
// Check plausibility 
IF f_InMax = f_InMin THEN	
	//
	// Not plausible output fix value
	F_ScalAnalogOut := 0;
ELSE	
	//
	// Plausible calculate output 
	f_DeltaIn:=f_InMax-f_InMin;
	f_DeltaOut:=f_OutMax-f_OutMin;
	F_ScalAnalogOut :=REAL_TO_INT((f_DeltaOut/f_DeltaIn)*(f_Input-f_InMin));	
END_IF

END_FUNCTION

// ---- POUs/P_Read_Research_Data.TcPOU
PROGRAM P_Read_Research_Data
VAR


END_VAR

//***********************************************************************************
//
// ETH Zürich / Robotic Fabrication Lab
// HIB C 13 / Stefano-Franscini-Platz 1
// CH-8093 Zürich
// 
// ***********************************************************************************
// 
// PROJECT     :  A061 Inline Mixer
// 
// FUNCTION    :  Read all research data for the process
// 
// AUTHOR      :  Seyma Gürel / Philippe Fleischmann
// 
// EMAIL       :  scotto@arch.ethz.ch / fleischmann@arch.ehtz.ch
// 
// Copyright   :  ETH Zürich (CH) 2021
//
// ***********************************************************************************


//
// Mixer run []
GVL_ResearchData.b_RED_Status_On:=GVL_VAR.b_MI1_Run;

//
// Mixer 1 speed override [%]
GVL_ResearchData.f_RED_Status_Speed_Overide:=GVL_VAR.f_MI1_Override;

//
// Mixer 1 current speed []
GVL_ResearchData.f_RED_Status_Speed_Motor_1:=GVL.Axis_Mixer1.NcToPlc.ActVelo;

//
// Mixer 1 current torque []
GVL_ResearchData.f_RED_Status_Torque_Motor_1:=GVL.f_MID1_ActTorque;

//
// Mixer 1 current motor temperature []
GVL_ResearchData.f_RED_Status_Temperature_Motor_1:=GVL.in_MID1_ActMotorTemperature *0.1; // weiting added 220817

//
// Mixer 2 current speed []
GVL_ResearchData.f_RED_Status_Speed_Motor_2:=GVL.Axis_Mixer1.NcToPlc.ActVelo;

//
// Mixer 2 current torque []
GVL_ResearchData.f_RED_Status_Torque_Motor_2:=GVL.f_MID2_ActTorque;

//
// Mixer 1 current motor temperature []
GVL_ResearchData.f_RED_Status_Temperature_Motor_2:=GVL.in_MID2_ActMotorTemperature *0.1; // weiting added 220817


//
// Accelration pump flowrate [ml/min]
GVL_ResearchData.f_RED_Status_Acceleration_Pump_Max_Flowrate_ml_per_min:=(GVL_ResearchData.f_RED_Acceleration_Pump_Mass/GVL_ResearchData.f_RED_Acceleration_Pump_Density);

END_PROGRAM

// ---- POUs/P_PP1_Ctrl_Manual.TcPOU
PROGRAM P_PP1_Ctrl_Manual
VAR
END_VAR

//***********************************************************************************
//
// ETH Zürich / Robotic Fabrication Lab
// HIB C 13 / Stefano-Franscini-Platz 1
// CH-8093 Zürich
// 
// ***********************************************************************************
// 
// PROJECT     :  A061 Inline Mixer
// 
// FUNCTION    :  Manual control of acceleration pump 1 
// 
// AUTHOR      :  Fabio Scotto / Philippe Fleischmann
// 
// EMAIL       :  scotto@arch.ethz.ch / fleischmann@arch.ehtz.ch
// 
// Copyright   :  ETH Zürich (CH) 2020
//
// ***********************************************************************************

//
// Place holder for manual control of the peristaltic pump 

;

END_PROGRAM

// ---- POUs/P_AP1_Ctrl_Manual.TcPOU
PROGRAM P_AP1_Ctrl_Manual

VAR

b_AP1_Error : BOOL;
b_AP1_Ready : BOOL;


END_VAR

//***********************************************************************************
//
// ETH Zürich / Robotic Fabrication Lab
// HIB C 13 / Stefano-Franscini-Platz 1
// CH-8093 Zürich
// 
// ***********************************************************************************
// 
// PROJECT     :  A061 Inline Mixer
// 
// FUNCTION    :  Manual control of peristaltic pump 
// 
// AUTHOR      :  Fabio Scotto / Philippe Fleischmann
// 
// EMAIL       :  scotto@arch.ethz.ch / fleischmann@arch.ehtz.ch
// 
// Copyright   :  ETH Zürich (CH) 2020
//
// ***********************************************************************************

//
// Place holder for manual control of the peristaltic pump 

//b_AP1_Error:=GVL_IO.ib_AP1_No_Error;
//b_AP1_Ready:=GVL_IO.ib_AP1_Ready;

//GVL_IO.ob_AP1_Power_On:=GVL_IO.ib_CC1_Button_Mode_Manual;
//GVL_IO.ob_AP1_Pressure_Ok:=TRUE;
//GVL_IO.ob_AP1_Not_Empty:=TRUE;
//GVL_IO.ob_AP1_Pulse:=FALSE;
//GVL_IO.ob_AP1_Start:=GVL_IO.ib_AP1_Button_On;

//GVL_IO.on_AP1_Speed:=GVL_IO.in_AP1_Poti_Speed;


;

END_PROGRAM
